FUNCTION TFGripperNearTilter : BOOL
VAR_INPUT
	PickPoint : TFMachinePalletizer_WorkPickPoint;
	Radius : LREAL;
	Modules : POINTER TO TFMachinePalletizer_Modules;
	
END_VAR
VAR
	Distance : LREAL;
END_VAR

TFGripperNearTilter := FALSE;

Distance := SQRT(((Modules^.Robot.XAx^.AxRef^.NcToPlc.ActPos-PickPoint.Xh)*(Modules^.Robot.XAx^.AxRef^.NcToPlc.ActPos-PickPoint.Xh))+
					((Modules^.Robot.YAx^.AxRef^.NcToPlc.ActPos-PickPoint.Yh)*(Modules^.Robot.YAx^.AxRef^.NcToPlc.ActPos-PickPoint.Yh))+
					((Modules^.Robot.ZAx^.AxRef^.NcToPlc.ActPos-PickPoint.Zh)*(Modules^.Robot.ZAx^.AxRef^.NcToPlc.ActPos-PickPoint.Zh)));


IF Distance <= Radius THEN
	TFGripperNearTilter := TRUE;
END_IF

END_FUNCTION

(* stored: Version 1.1.0.1, ProductVersion 3.1.4024.11
   POU TFGripperNearTilter: Id {18aa30e6-ffd4-4084-929a-b15a4f17b2e1}, SpecialFunc None *)
